(* LS Electric XG5000 project: OUTNAT1 *)
(* PLC LSPLC *)

PROGRAM NewProgram (* task: 스캔 프로그램 *)

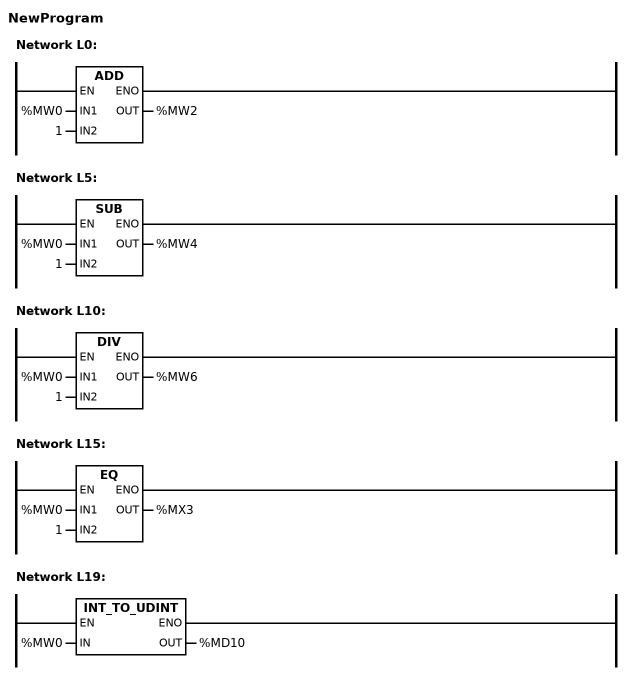
(* Rung L0 *)
%MW2 := %MW0 + 1;
(* Rung L5 *)
%MW4 := %MW0 - 1;
(* Rung L10 *)
%MW6 := %MW0 / 1;
(* Rung L15 *)
%MX3 := %MW0 = 1;
(* Rung L19 *)
%MD10 := INT_TO_UDINT(%MW0);
END_PROGRAM